{attribute 'linkalways'} 
{attribute 'no_explicit_call' := 'This FB is a CLASS and must be accessed using methods or properties'}
{attribute 'enable_dynamic_creation'}
FUNCTION_BLOCK _TcVnImageInfo EXTENDS StructuredDatatypeBase
VAR
	localData : TcVnImageInfo;
	activeData : REFERENCE TO TcVnImageInfo REF= localData;
	_nImageSize : _ULINT(localData.nImageSize);
	_nWidth : _UDINT(localData.nWidth);
	_nHeight : _UDINT(localData.nHeight);
	_nXPadding : _UINT(localData.nXPadding);
	_nYPadding : _UINT(localData.nYPadding);
	_stPixelFormat : _TcVnPixelFormat();
END_VAR

PROPERTY PUBLIC Address : PVOID
GET
Address := ADR(activeData);
END_GET
END_PROPERTY

METHOD PUBLIC ClearReference
VAR_INPUT
END_VAR
activeData REF= localData;
SetMemberReference();
END_METHOD

METHOD PUBLIC Clone : I_Datatype
VAR
    pClone : POINTER TO _TcVnImageInfo;
END_VAR
pClone := __NEW(_TcVnImageInfo());
pClone^.Value := Value;
Clone := pClone^;
END_METHOD

METHOD FB_init : BOOL
VAR_INPUT
	bInitRetains : BOOL; // if TRUE, the retain variables are initialized (warm start / cold start)
	bInCopyCode : BOOL;  // if TRUE, the instance afterwards gets moved into the copy code (online change)
END_VAR
SetMemberReference();
AddMember('nImageSize',_nImageSize);
AddMember('nWidth',_nWidth);
AddMember('nHeight',_nHeight);
AddMember('nXPadding',_nXPadding);
AddMember('nYPadding',_nYPadding);
AddMember('stPixelFormat',_stPixelFormat);
END_METHOD

PROPERTY PUBLIC Identifier : T_MAXSTRING
GET
Identifier := 'TcVnImageInfo';
END_GET
END_PROPERTY

METHOD PUBLIC MakeReferenceTo
VAR_INPUT
	ReferenceTarget : REFERENCE TO TcVnImageInfo;
END_VAR
activeData REF= ReferenceTarget;
SetMemberReference();
END_METHOD

PROPERTY PUBLIC nHeight : Reference to _UDINT
GET
nHeight REF= _nHeight;
END_GET
END_PROPERTY

PROPERTY PUBLIC nImageSize : Reference to _ULINT
GET
nImageSize REF= _nImageSize;
END_GET
END_PROPERTY

PROPERTY PUBLIC nWidth : Reference to _UDINT
GET
nWidth REF= _nWidth;
END_GET
END_PROPERTY

PROPERTY PUBLIC nXPadding : Reference to _UINT
GET
nXPadding REF= _nXPadding;
END_GET
END_PROPERTY

PROPERTY PUBLIC nYPadding : Reference to _UINT
GET
nYPadding REF= _nYPadding;
END_GET
END_PROPERTY

METHOD PROTECTED SetMemberReference
VAR_INPUT
END_VAR
_nImageSize.MakeReferenceTo(activeData.nImageSize);
_nWidth.MakeReferenceTo(activeData.nWidth);
_nHeight.MakeReferenceTo(activeData.nHeight);
_nXPadding.MakeReferenceTo(activeData.nXPadding);
_nYPadding.MakeReferenceTo(activeData.nYPadding);
_stPixelFormat.MakeReferenceTo(activeData.stPixelFormat);
END_METHOD

PROPERTY PUBLIC Size : UDINT
GET
Size := SIZEOF(activeData);
END_GET
END_PROPERTY

PROPERTY PUBLIC stPixelFormat : Reference to _TcVnPixelFormat
GET
stPixelFormat REF= _stPixelFormat;
END_GET
END_PROPERTY

METHOD TryMakeReferenceTo : BOOL
VAR_INPUT
	Target : I_Datatype;
END_VAR
VAR
	targetAsStruct : I_StructuredDatatype;
	pTargetData : POINTER TO TcVnImageInfo;
END_VAR
IF NOT Target.TryResolveAsStructuredDatatype(targetAsStruct) THEN
	RETURN;
END_IF

IF NOT (targetAsStruct.Identifier = Identifier) THEN
	RETURN;
END_IF

pTargetData := Target.Address;
activeData REF= pTargetData^;
SetMemberReference();
TryMakeReferenceTo := TRUE;
END_METHOD

PROPERTY PUBLIC Value : REFERENCE TO TcVnImageInfo
GET
Value REF= activeData;
END_GET
END_PROPERTY

END_FUNCTION_BLOCK

(* stored: Version 1.1.0.1, ProductVersion 3.1.4024.13
   POU _TcVnImageInfo: Id {b656643e-378b-481c-83e1-1039eda8cdca}, SpecialFunc None
   Folder Constructor: Id {f45b398f-6ee9-4753-85b3-1559cf197c26}
   Folder Protected: Id {ea45eedf-6f26-46ba-988d-9f2634667521}
   Property Address: Id {e80dff28-19f0-44df-8834-8266fbb092a1}
   Get Get: Id {3f161686-c595-403b-9102-16372805bce8}
   Method ClearReference: Id {7f85774e-74a5-43d4-a61e-54a24641ec41}
   Method Clone: Id {66294728-a3e0-4735-9a0b-5998a2f8ce03}
   Method FB_init: Id {8d1040ae-323a-4611-8306-d933e0555047}
   Property Identifier: Id {61386bb3-a6fe-4bcd-9e25-9cc995fdff8f}
   Get Get: Id {71c0a82a-6e05-4713-a11c-7292bdaa2c05}
   Method MakeReferenceTo: Id {721a83af-1cb7-4713-9de1-50c38dad631d}
   Property nHeight: Id {c2628e39-f5ca-40e1-bdaa-bdcc9f31c12b}
   Get Get: Id {554634f8-da37-446c-b7ff-51ae37f1dd13}
   Property nImageSize: Id {eec93768-9d1a-459a-90ee-3373438e72f7}
   Get Get: Id {7cc52221-d7f5-48b3-adfa-8c560c4ada00}
   Property nWidth: Id {e0933265-78ec-4dd9-bfad-78b5c93275b5}
   Get Get: Id {aa717872-7dde-4d1e-80db-63a979398962}
   Property nXPadding: Id {c8c7fd79-aa62-4d6b-9afc-6a26f96c17d3}
   Get Get: Id {fd6a59fe-c273-4905-96ce-0ae8c89967b9}
   Property nYPadding: Id {bde01df4-53f1-49ef-ab5e-9a8f204913f9}
   Get Get: Id {1d477318-0c76-4d5b-a79e-00c3e64f0d2c}
   Method SetMemberReference: Id {460b2126-61aa-4748-9dd3-525c5417c9a1}
   Property Size: Id {721f4d0a-b644-4b6c-b947-daedec0f4eb7}
   Get Get: Id {072bc006-dd78-4dff-8a03-6bcb65bd86c6}
   Property stPixelFormat: Id {8a5a2d79-3c92-4df4-bad0-1fcd8c057252}
   Get Get: Id {be3f8677-6d62-4aad-a120-f17e745f5e46}
   Method TryMakeReferenceTo: Id {10586b83-7455-4d67-a741-87f66a63e043}
   Property Value: Id {f9d166eb-9019-40ec-9f45-a443665f9b35}
   Get Get: Id {0a6fbf2a-93f8-427c-9062-f928f44d42d1} *)
